Universal Robots PolyScope program: RC_E3_MOVE_310.urp

Program RC_E3_MOVE_310 (createdIn=3.0.0 lastSavedIn=3.0.0 directory=/programs installation=default)
Robot Program (runOnlyOnce=true motionType=MoveJ speed=1.047198 acceleration=1.396263 useActiveTCP=false)
  'Program generated by RoboDK v4.1.0 for UR3e_HORNO on 27/07/2022 12:02:44'
  'Using nominal kinematics.'
  'Using Ref. UR3_2: p[0.000000, 0.000000, 0.000000, 0.000000, 0.000000, 0.000000]'
  'Using TCP 0208-0001-0001-307-000-3 Horno: p[0.000000, 0.000000, 0.038000, 0.000000, 0.000000, 0.000000]'
  Script: set_tcp(p[0.000000, 0.000000, 0.038000, 0.000000, 0.000000, 0.000000])
  Script: movej([1.639213, -1.273043, -1.014734, -0.852942, 1.521404, 0.000000],0.60000,0.12500,0,0.0000)
